(* CoDeSys 2.3.9.59 project: CLIMAVIN_exempleHoraires.pro *)
(* Libraries: Standard.lib, Util.lib 20.3.15 11:30:08, SysLibCallback.lib, SysLibSockets.lib, SysLibTasks.lib, SysLibRtc.lib, SysLibFile.lib, SysLibPlcCtrl.lib, SysLibRtc_Add.lib, easy800_gb.lib 3.8.10 12:23:32, SysLibTime.lib *)

(* POU PLC_PRG, ST *)
PROGRAM PLC_PRG
VAR
	fbTimeManagement01: HW;		(*Bloc fonction horaires*)
	fbTimeManagement02: HW;		(*Bloc fonction horaires*)
	xFbOut01: BOOL;				(*Sortie du bloc 01*)
	xFbOut02: BOOL;				(*Sortie du bloc 02*)
	dtCurrentDateAndTime: DT;
	dummy: BOOL;
END_VAR
(*=================================================================================================
	Programme exemple de gestion d'horaires sur une semaine
===================================================================================================
	Nom :		CLIMAVIN_exempleHoraires
	Date :		14/05/2024
	Version :	V1.0.0
	Matériel :	XV300
	CoDeSys :	V2.3.9 SP8
	Auteur :	Bruno COTTANCIN
===================================================================================================
	Librairies :
		- easy800_gb.lib
===================================================================================================
	NOTE IMPORTANTE
	~~~~~~~~~~~~~~~
		Nous vous rappellons que ceci est un exemple de programme dont l’objectif est de vérifier
		le bon fonctionnement de l’application.
		Vous pouvez utiliser cet exemple de programme mais nous vous conseillons de tester son
		fonctionnement dans des conditions qui NE mettront pas l’installation en péril.
		La mise en śuvre et l’exploitation de ce programme sont sous votre responsabilité.
=================================================================================================*)


(* === heure courante (pour info) === *)

dtCurrentDateAndTime := SysRtcGetTime(dummy);


(* === gestion d'horaires 2 premiers jours === *)

fbTimeManagement01(			(* Gestion deux canaux (A et B) *)
	EN		:= TRUE,
	A_DY1	:= Mo,			(* 1er canal (A) du lundi au lundi *)
	A_DY2	:= Mo,
	A_ON_h	:= 8,			(* de 8:00 ŕ 18:00 *)
	A_ON_m	:= 0,
	A_OFF_h	:= 18,
	A_OFF_m	:= 0,
	B_DY1	:= Tu,			(* 2nd canal (B) du mardi au mardi *)
	B_DY2	:= Tu,
	B_ON_h	:= 9,			(* de 9:15 ŕ 19:37 *)
	B_ON_m	:= 15,
	B_OFF_h	:= 19,
	B_OFF_m	:= 37,
	Q1		=> xFbOut01
);


(* === gestion d'horaires 2 autres jours === *)

fbTimeManagement02(			(* Gestion deux canaux (A et B) *)
	EN		:= TRUE,
	A_DY1	:= We,			(* 1er canal (A) du mercredi au mercredi *)
	A_DY2	:= We,
	A_ON_h	:= 7,			(* de 7:10 ŕ 17:20 *)
	A_ON_m	:= 10,
	A_OFF_h	:= 17,
	A_OFF_m	:= 20,
	B_DY1	:= Th,			(* 2nd canal (B) du jeudi au jeudi *)
	B_DY2	:= Th,
	B_ON_h	:= 8,			(* de 8:12 ŕ 21:12 *)
	B_ON_m	:= 12,
	B_OFF_h	:= 21,
	B_OFF_m	:= 12,
	Q1		=> xFbOut02
);


(* Etc... *)
END_PROGRAM
